{attribute 'linkalways'} 
{attribute 'no_explicit_call' := 'This FB is a CLASS and must be accessed using methods or properties'}
{attribute 'enable_dynamic_creation'}
FUNCTION_BLOCK Promise EXTENDS Disposable IMPLEMENTS I_Promise
VAR
	context : PromiseContext;
END_VAR

PROPERTY PUBLIC Ctx : I_PromiseContext
GET
Ctx := context;
END_GET
END_PROPERTY

PROPERTY PUBLIC Pending : BOOL
GET
Pending := context.Pending;
END_GET
END_PROPERTY

PROPERTY Rejected : BOOL
GET
Rejected := context.Rejected;
END_GET
END_PROPERTY

PROPERTY RejectedReason : T_MAXSTRING
GET
RejectedReason := context.RejectedReason;
END_GET
END_PROPERTY

PROPERTY Resolved : BOOL
GET
Resolved := context.Resolved;
END_GET
END_PROPERTY

METHOD PUBLIC TryGetResult : BOOL
VAR_INPUT
	Destination : ANY;
END_VAR
TryGetResult := context.TryGetResult(Destination);
END_METHOD

METHOD PUBLIC TryGetResultTo : BOOL
VAR_INPUT
	DestinationAddress : PVOID;
	DestinationSize : UDINT;
END_VAR
TryGetResultTo := context.TryGetResultTo(DestinationAddress,DestinationSize);
END_METHOD

END_FUNCTION_BLOCK

(* stored: Version 1.1.0.1
   POU Promise: Id {03f37619-5178-475e-a9f8-676071412171}, SpecialFunc None
   Property Ctx: Id {d99e08bb-f6d7-481a-b8d4-3d55da41d317}
   Get Get: Id {918dbfb4-df26-400e-8685-a4e46781d6d9}
   Property Pending: Id {dc75c018-e00f-4422-9140-9bcf7c1277fd}
   Get Get: Id {204e0cfa-0241-4c1d-835a-6a3c59935bc4}
   Property Rejected: Id {c56b3631-f2a9-4af7-8b2b-35078f245833}
   Get Get: Id {86bc78af-a066-497b-810b-8a0910718fb6}
   Property RejectedReason: Id {be210ed0-dbf1-4088-893e-3ed986b72f13}
   Get Get: Id {c5e08e5b-a914-4aa9-a0e9-a821e31a9ef2}
   Property Resolved: Id {10e6266d-e498-41b8-87e3-34372768f2e0}
   Get Get: Id {114c3428-4438-44f0-a7c0-fc9fc89ccdd2}
   Method TryGetResult: Id {729c3634-87d6-440e-bf59-06cb9e843967}
   Method TryGetResultTo: Id {f332e9b6-bb5b-49c8-8390-c2fb5200ec9c} *)
